// TIA Portal V19 export
FUNCTION_BLOCK "Temperature_Control_Concurant"   // FB19, LAD
{ S7_Optimized_Access := 'TRUE' }
// stored: MemoryReserve 100, SetENOAutomatically false
   VAR_INPUT
      Enable : Bool;
      "Temperature Sensor" : Real;
      "Process Values" : Array[0..1] of Real;
      "Main Valve Max Temperature" : Real;
      "simmer offset" : Real;
      "Jacket or Lance" : Bool;
      "auto Run EN" : Bool;
   END_VAR
   VAR_OUTPUT
      "Main Valve" : Bool;
      "Simmer Valve" : Bool;
      Running : Bool;
      "Enable Valve" : Bool;
      "Holding Temperature" : Bool;
      "Run Constant" : Bool;
      "Step Completed" : Bool;
   END_VAR
   VAR
      "Main Valve SP" : Real;
      "Main Valve SP Reached" : Bool;
      IEC_Timer_0_Instance { S7_SetPoint := 'True'} : TON_TIME;
      IEC_Timer_0_Instance_1 { S7_SetPoint := 'True'} : TON_TIME;
   END_VAR
BEGIN

REGION Network 1
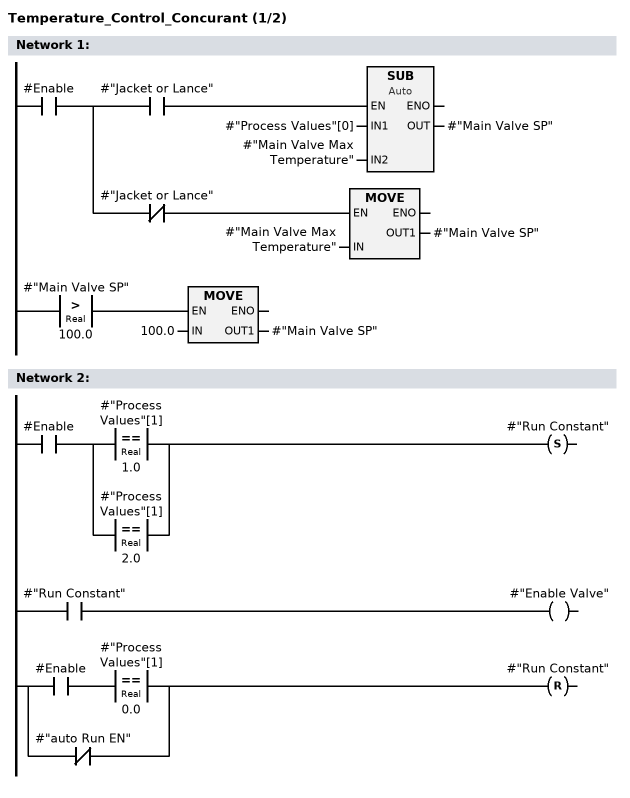
   RUNG wire#powerrail
      Contact( #Enable )
      wire#w1
      Contact( #"Jacket or Lance" )
      Sub(in1 := #"Process Values"[0], in2 := #"Main Valve Max Temperature", out => #"Main Valve SP")
   END_RUNG
   RUNG wire#w1
      I_Contact( #"Jacket or Lance" )
      Move(in := #"Main Valve Max Temperature", out1 => #"Main Valve SP")
   END_RUNG
   RUNG wire#powerrail
      { S7_Templates := "SrcType := Real" } GT_Contact(in1 := #"Main Valve SP", in2 := 100.0)
      Move(in := 100.0, out1 => #"Main Valve SP")
   END_RUNG
   // the same network as SCL:
   IF #Enable AND #"Jacket or Lance" THEN
       #"Main Valve SP" := #"Process Values"[0] - #"Main Valve Max Temperature";
   END_IF;
   IF #Enable AND NOT #"Jacket or Lance" THEN #"Main Valve SP" := #"Main Valve Max Temperature"; END_IF;
   IF #"Main Valve SP" > 100.0 THEN #"Main Valve SP" := 100.0; END_IF;
END_REGION

REGION Network 2
   RUNG wire#powerrail
      Contact( #Enable )
      wire#w1
      { S7_Templates := "SrcType := Real" } EQ_Contact(in1 := #"Process Values"[1], in2 := 1.0)
      wire#w2
      S_Coil( #"Run Constant" )
   END_RUNG
   RUNG wire#w1
      { S7_Templates := "SrcType := Real" } EQ_Contact(in1 := #"Process Values"[1], in2 := 2.0)
   END_RUNG wire#w2
   RUNG wire#powerrail
      Contact( #"Run Constant" )
      Coil( #"Enable Valve" )
   END_RUNG
   RUNG wire#powerrail
      Contact( #Enable )
      { S7_Templates := "SrcType := Real" } EQ_Contact(in1 := #"Process Values"[1], in2 := 0.0)
      wire#w3
      R_Coil( #"Run Constant" )
   END_RUNG
   RUNG wire#powerrail
      I_Contact( #"auto Run EN" )
   END_RUNG wire#w3
   // the same network as SCL:
   IF #Enable AND ((#"Process Values"[1] = 1.0) OR (#"Process Values"[1] = 2.0)) THEN
       #"Run Constant" := TRUE;
   END_IF;
   #"Enable Valve" := #"Run Constant";
   IF (#Enable AND (#"Process Values"[1] = 0.0)) OR NOT #"auto Run EN" THEN #"Run Constant" := FALSE; END_IF;
END_REGION

REGION Network 3
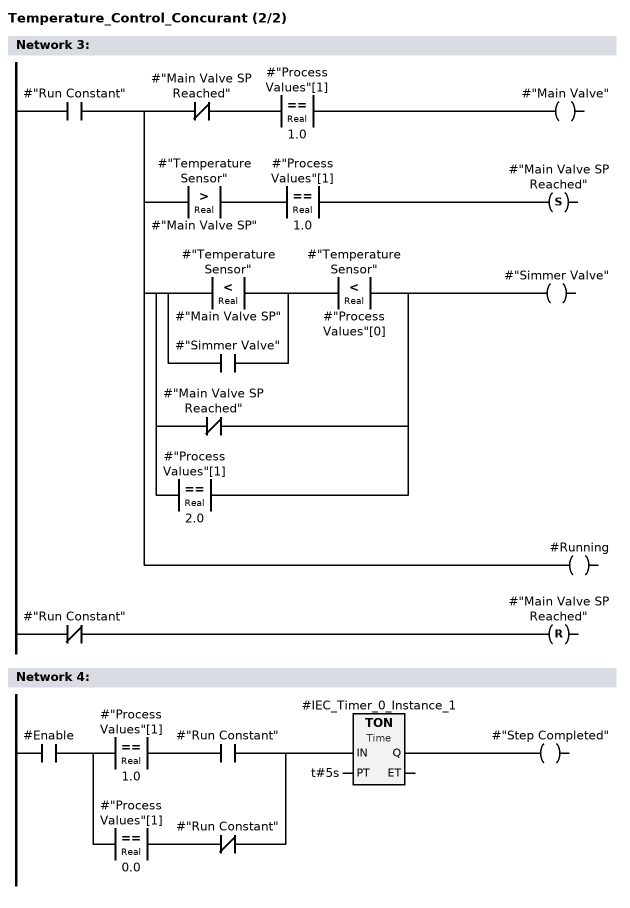
   RUNG wire#powerrail
      Contact( #"Run Constant" )
      wire#w1
      I_Contact( #"Main Valve SP Reached" )
      { S7_Templates := "SrcType := Real" } EQ_Contact(in1 := #"Process Values"[1], in2 := 1.0)
      Coil( #"Main Valve" )
   END_RUNG
   RUNG wire#w1
      { S7_Templates := "SrcType := Real" } GT_Contact(in1 := #"Temperature Sensor", in2 := #"Main Valve SP")
      { S7_Templates := "SrcType := Real" } EQ_Contact(in1 := #"Process Values"[1], in2 := 1.0)
      S_Coil( #"Main Valve SP Reached" )
   END_RUNG
   RUNG wire#w1
      { S7_Templates := "SrcType := Real" } LT_Contact(in1 := #"Temperature Sensor", in2 := #"Main Valve SP")
      wire#w2
      { S7_Templates := "SrcType := Real" } LT_Contact(in1 := #"Temperature Sensor", in2 := #"Process Values"[0])
      wire#w3
      Coil( #"Simmer Valve" )
   END_RUNG
   RUNG wire#w1
      Contact( #"Simmer Valve" )
   END_RUNG wire#w2
   RUNG wire#w1
      I_Contact( #"Main Valve SP Reached" )
   END_RUNG wire#w3
   RUNG wire#w1
      { S7_Templates := "SrcType := Real" } EQ_Contact(in1 := #"Process Values"[1], in2 := 2.0)
   END_RUNG wire#w3
   RUNG wire#w1
      Coil( #Running )
   END_RUNG
   RUNG wire#powerrail
      I_Contact( #"Run Constant" )
      R_Coil( #"Main Valve SP Reached" )
   END_RUNG
   // the same network as SCL:
   #"Main Valve" := #"Run Constant" AND NOT #"Main Valve SP Reached" AND (#"Process Values"[1] = 1.0);
   IF #"Run Constant" AND (#"Temperature Sensor" > #"Main Valve SP") AND (#"Process Values"[1] = 1.0) THEN
       #"Main Valve SP Reached" := TRUE;
   END_IF;
   #"Simmer Valve" := #"Run Constant" AND ((((#"Temperature Sensor" < #"Main Valve SP") OR #"Simmer Valve") AND (#"Temperature Sensor" < #"Process Values"[0])) OR NOT #"Main Valve SP Reached" OR (#"Process Values"[1] = 2.0));
   #Running := #"Run Constant";
   IF NOT #"Run Constant" THEN #"Main Valve SP Reached" := FALSE; END_IF;
END_REGION

REGION Network 4
   RUNG wire#powerrail
      Contact( #Enable )
      wire#w1
      { S7_Templates := "SrcType := Real" } EQ_Contact(in1 := #"Process Values"[1], in2 := 1.0)
      Contact( #"Run Constant" )
      wire#w2
      { S7_Templates := "time_type := Time" } #IEC_Timer_0_Instance_1.TON(pt := t#5s, et =>)
      Coil( #"Step Completed" )
   END_RUNG
   RUNG wire#w1
      { S7_Templates := "SrcType := Real" } EQ_Contact(in1 := #"Process Values"[1], in2 := 0.0)
      I_Contact( #"Run Constant" )
   END_RUNG wire#w2
   // the same network as SCL:
   #IEC_Timer_0_Instance_1(IN := #Enable AND (((#"Process Values"[1] = 1.0) AND #"Run Constant") OR ((#"Process Values"[1] = 0.0) AND NOT #"Run Constant")),   // TON
                           PT := t#5s);
   #"Step Completed" := #IEC_Timer_0_Instance_1.Q;
END_REGION
END_FUNCTION_BLOCK
